VAR_GLOBAL
	itf_content : ST_adsITF;			
END_VAR

(* stored: Version 1.1.0.1, ProductVersion 3.1.4024.11
   GVL GVL_adsITF: Id {39d11898-66da-4a0a-9531-37a3dec525bf} *)
